// TIA Portal V16 export
// export: Created 2021-07-12T14:47:20.4387518Z, ExportSetting WithDefaults, DisplayName Totally Integrated Automation Portal, DisplayVersion V16, DisplayName TIA Portal Version Control Interface, DisplayVersion V16, DisplayName TIA Portal Openness, DisplayVersion V16, DisplayName STEP 7 Professional, DisplayVersion V16, DisplayName STEP 7 Safety, DisplayVersion V16, DisplayName WinCC Professional, DisplayVersion V16
TYPE "SimaHydTO_typeVCharArray"
TITLE = SimaHydTO_typeVCharArray
// VChar (characteristics) array of HMI VChar selection
// stored: IsFailsafeCompliant false
   STRUCT
      VChar_DB : DB_ANY;   // DB number of VChar storage
      measurementConfig { S7_SetPoint := 'True'} : "LSimaHydTO_typeMeasurementConfig";
      initialized : Bool;
   END_STRUCT;
END_TYPE
